FUNCTION_BLOCK FB_PendantControl
VAR_INPUT
	fbCovers			: I_MirrorCovers;
	fbBrake				: I_Brake;
	fbHydraulics		: I_Hydraulics;
	fbFocus		 		: I_Focus;
	fbElevation			: REFERENCE TO FB_ElevationControl;
	fbAzimuth	 		: REFERENCE TO FB_AzimuthControl;
	fbDerotator			: REFERENCE TO FB_DerotatorControl;
	fbTelescope			: REFERENCE TO FB_TelescopeControl;	
END_VAR
VAR
	comm				: I_Comm;

	// program selection of the pendant control
	Selection:	UINT;
	// error on the pendant control
	Error:		BOOL;
	horn:			BOOL;
	fbStartTrigger			: R_TRIG;
	DerotatorEnable:	FB_ButtonEnable;
	ElevationEnable: 	FB_ButtonEnable;
	AzimuthEnable: 		FB_ButtonEnable;
	TelescopeControlEnable: 	FB_ButtonEnable;
	TrackingEnable:			FB_ButtonEnable;
	ResetDelay:	TON;
	TwinCATRestart: TC_Restart;
	up_trigger:	R_TRIG;
	down_trigger:	R_TRIG;	
	// manual or automatic operation of the telescope
	telescope_mode : E_TelescopeMode;
	
	reset_trigger		: R_TRIG;

	//DIN17 2.0
	BCD0		AT%I*: BOOL;
	//DIN18 2.1
	BCD2		AT%I*: BOOL;
	//DIN19 2.2
	BCD4		AT%I*: BOOL;
	//DIN20 2.3
	BCD8		AT%I*: BOOL;
	//DIN21 2.4
	reset_switch	AT%I*: BOOL;
	//DIN22 2.5
	direction_up	AT%I*: BOOL;
	//DIN23 2.6
	direction_down	AT%I*: BOOL;
	//DIN24 2.7
	key_switch		AT%I*: BOOL;
	//DIN25 3.0 (enable)
	start_switch	AT%I*: BOOL;
	//DIN26 3.1
	direction_left	AT%I*: BOOL;
	//DIN27 3.2
	direction_right	AT%I*: BOOL;
	
	// Outputs
	
	//DOUT9 1.0
	lamp_up			AT%Q*: BOOL;
	//DOUT10 1.1
	lamp_down			AT%Q*: BOOL;
	//DOUT11 1.2
	lamp_right			AT%Q*: BOOL;
	//DOUT12 1.3
	lamp_left			AT%Q*: BOOL;
	//DOUT13 1.4
	lamp_error			AT%Q*: BOOL;	
END_VAR

(* 
This program is responsible for the manual control of the telescope.
all movable parts can be controlled from here. This is mainly for testing and
maintenance.
WARNING! Some of the safety routines are disabled, when operating the telescope manually.
*)
// calculate the value of the selector
Selection := 1*BOOL_TO_UINT(BCD0) + 
			 2*BOOL_TO_UINT(BCD2) + 
			 4*BOOL_TO_UINT(BCD4) +
			 8*BOOL_TO_UINT(BCD8);

// detect disconnection of the manual controls (should also trigger emergency stop).			 
Error := (Selection = 0);

// disable all the lamps
lamp_left := FALSE;
lamp_right := FALSE;
lamp_up := FALSE;
lamp_down := FALSE;
horn := FALSE;

up_trigger(CLK := direction_up);
down_trigger(CLK := direction_down);
//R_Enable(CLK := enable);
// the error lamp is the same as the error lamp of the main panel
lamp_error := lamp_error;


// determine the operation of the telescope based on the switch set
IF key_switch THEN
	telescope_mode := E_TelescopeMode.manual;
ELSE
	telescope_mode := E_TelescopeMode.automatic;
END_IF

// reset or start pushed?
reset_trigger(CLK := reset_switch);
fbStartTrigger(CLK := start_switch);

// enable only the selected item and connect lamps and buttons accordingly
CASE Selection OF
	1, 2, 3:	// reserved for Cover 1-3 control
		lamp_up := fbCovers.IsCoverOpen(Selection);
		lamp_down := fbCovers.IsCoverClosed(Selection);
		IF key_switch THEN
			IF direction_up AND fbCovers.IsCoverOpen(Selection) THEN
				fbCovers.OpenCover(Selection);
			ELSIF direction_down AND fbCovers.IsCoverClosed(Selection) THEN
				fbCovers.CloseCover(Selection);
			END_IF
			lamp_error := fbCovers.HasError(Selection);	
		ELSE
			IF direction_down THEN 
				fbCovers.CloseCovers();
			ELSIF direction_up THEN
				fbCovers.OpenCovers();
			END_IF		
		END_IF
		
	4:	// Nasmyth / mirror M3 control
		
	5:	// Focus Control
		IF fbFocus <> 0 THEN
			lamp_up := fbFocus.Ready AND NOT fbFocus.InFarLimit;
			lamp_down := fbFocus.Ready AND NOT fbFocus.InNearLimit;
			IF key_switch THEN
				IF fbStartTrigger.Q THEN
					fbFocus.Enable := NOT fbFocus.Enable;
				END_IF
				fbFocus.MoveOut(direction_up);
				fbFocus.MoveIn(direction_down);
				IF reset_trigger.Q THEN
					fbFocus.Reset();
				END_IF
				lamp_error := fbFocus.Error;
			END_IF
		END_IF
							
	6:	// Derotator control
		lamp_left  := fbDerotator.IsReady() AND NOT fbDerotator.IsInMinLimit();
		lamp_right := fbDerotator.IsReady() AND NOT fbDerotator.IsInMaxLimit();
		IF key_switch THEN
			DerotatorEnable(SET := start_switch, Q := fbDerotator.bEnable);
			fbDerotator.MoveLeft(direction_left AND NOT fbDerotator.inDigitalInputs.1);
			fbDerotator.MoveRight(direction_right AND NOT fbDerotator.inDigitalInputs.0);
			fbDerotator.bReset := reset_switch;
			lamp_error := fbDerotator.bError;
		END_IF
							
	7:	// Elevation Control
		
		fbElevation.bUp := direction_up AND fbElevation.inDigitalInputs.0;
		fbElevation.bDown := direction_down AND fbElevation.inDigitalInputs.1;
		IF key_switch THEN
			ElevationEnable(
				SET := start_switch, 
				Q := fbElevation.bEnable);	
		END_IF
		fbElevation.bReset := reset_switch;
		lamp_up := fbElevation.inDigitalInputs.0;
		lamp_down := fbElevation.inDigitalInputs.1;
		lamp_error := fbElevation.bError;
		
	8:	// Azimuth Control
		lamp_left := fbAzimuth.inDigitalInputs.0; // NOT GVL_Telescope.azimut_limit_switch;
		lamp_right := fbAzimuth.inDigitalInputs.1; // NOT GVL_Telescope.azimut_limit_switch;
		fbAzimuth.bLeft := direction_left AND fbAzimuth.inDigitalInputs.0;
		fbAzimuth.bRight := direction_right AND fbAzimuth.inDigitalInputs.1;
		fbAzimuth.bReset := reset_switch;
		IF key_switch THEN
			AzimuthEnable(
				SET := start_switch, 
				Q := fbAzimuth.bEnable);
			lamp_error := fbAzimuth.bError;
		END_IF
		
	9: 	// Dome control
		
	10:	// FilterWheel control
		
	11: lamp_up := fbElevation.fTorque > 0.0;
		lamp_down := fbElevation.fTorque < 0.0;
		
	12:	// manual Telescope Control
		IF key_switch THEN
			lamp_up := fbTelescope.power;
			lamp_down := fbTelescope.power;
			lamp_left := fbTelescope.power;
			lamp_right := fbTelescope.power;
	
			fbTelescope.gohome := direction_down;
			fbTelescope.park := direction_up;
			fbTelescope.goto := direction_right;
			TrackingEnable(SET := start_switch, 
							RESET := reset_switch, 
							Q := fbTelescope.track);
			fbTelescope.reset := reset_switch;
			fbTelescope.stop := direction_left;	
			lamp_error := fbTelescope.error;
		END_IF
		
	13: // Telescope Control
		TelescopeControlEnable(
			SET := start_switch, 
			Q := fbTelescope.power);
		fbTelescope.reset := reset_switch;
		IF key_switch THEN
			lamp_up := fbElevation.inDigitalInputs.0;
			lamp_down := fbElevation.inDigitalInputs.1;
			lamp_left := fbAzimuth.inDigitalInputs.0;
			lamp_right := fbAzimuth.inDigitalInputs.1;
			fbElevation.bUp := direction_up AND fbElevation.inDigitalInputs.0;
			fbElevation.bDown := direction_down AND fbElevation.inDigitalInputs.1;
			fbAzimuth.bLeft := direction_left AND fbAzimuth.inDigitalInputs.0;
			fbAzimuth.bRight := direction_right AND fbAzimuth.inDigitalInputs.1;
			fbTelescope.rightascension := fbTelescope.rightascension_calc;
			fbTelescope.declination := fbTelescope.declination_calc;
		ELSE
			lamp_up := fbElevation.bEnable;
			lamp_down := fbElevation.bEnable;
			lamp_left := fbAzimuth.bEnable;
			lamp_right := fbAzimuth.bEnable;
			IF direction_up THEN 
				fbTelescope.elevation_offset := fbTelescope.elevation_offset + 10.0/3600.0; 
			ELSIF direction_down THEN 
				fbTelescope.elevation_offset := fbTelescope.elevation_offset - 10.0/3600.0; 
			END_IF;
			IF direction_left THEN 
				fbTelescope.azimuth_offset := fbTelescope.azimuth_offset - 10.0/3600.0; 
			ELSIF direction_right THEN 
				fbTelescope.azimuth_offset := fbTelescope.azimuth_offset + 10.0/3600.0; 
			END_IF;
		END_IF
		ResetDelay(IN := reset_switch, PT := T#3S);
		// wait for suction pump to stop
		TwinCATRestart(NETID := '', RESTART := ResetDelay.Q AND NOT fbHydraulics.SuctionRunning, TMOUT := T#60S);
	
	14: horn := key_switch;
		lamp_up := key_switch;
		lamp_down := key_switch;
		lamp_left := key_switch;
		lamp_right := key_switch;
	
	15:	// Hydraulics control
		lamp_up := fbHydraulics.OilPressureOK AND NOT fbBrake.BrakeOpen;
		lamp_down := fbHydraulics.OilPressureOK AND fbBrake.BrakeOpen;
		lamp_left := fbHydraulics.PumpRunning;
		lamp_right := fbHydraulics.SuctionRunning;
		IF key_switch THEN
			IF fbStartTrigger.Q THEN
				fbHydraulics.Enable := NOT fbHydraulics.Enable;
			END_IF
			IF reset_trigger.Q THEN
				fbHydraulics.Reset();
			END_IF
			
			IF direction_up THEN
				fbBrake.OpenBrake();
			END_IF
			IF direction_down THEN
				fbBrake.CloseBrake();
			END_IF
			fbHydraulics.ManualStartSuction := direction_right;
			fbHydraulics.ManualStopPump := direction_left;
			lamp_error := fbHydraulics.Error;
		END_IF
END_CASE

//FB_Init is always available implicitly and it is used primarily for initialization.
//The return value is not evaluated. For a specific influence, you can also declare the
//methods explicitly and provide additional code there with the standard initialization
//code. You can evaluate the return value.
METHOD FB_Init: BOOL
VAR_INPUT
    bInitRetains: BOOL; // TRUE: the retain variables are initialized (reset warm / reset cold)
    bInCopyCode: BOOL;  // TRUE: the instance will be copied to the copy code afterward (online change)
	comm			: I_Comm;   
END_VAR
THIS^.comm 	:= comm;
END_METHOD

END_FUNCTION_BLOCK

(* stored: Version 1.1.0.1, ProductVersion 3.1.4026.11
   POU FB_PendantControl: Id {e2b10f6c-d16d-4403-9ebe-8d8a369c8dbd}, SpecialFunc None
   Method FB_Init: Id {377c4b19-44fb-4929-801b-86205f66218e} *)
